FUNCTION_BLOCK Eventlogger
VAR
	Eventbuffer: ARRAY [1..MAXIMUM_NUMBER_OF_EVENTS] OF ST_Event;
	CurrentEventNumber : INT :=0;
	_PersistentEventStorage: I_PersistentStorage;
	
END_VAR
VAR CONSTANT
	MAXIMUM_NUMBER_OF_EVENTS: INT:=100;
END_VAR

METHOD PUBLIC AddEvent : BOOL
VAR_INPUT
	eEventType: E_EventType;
	eEventSeverity: TcEventSeverity;
	nEventIdentity: UDINT;
	sEventText: STRING(255);
END_VAR
IF NOT IsEventBufferFull() THEN
		CurrentEventNumber := CurrentEventNumber +1;
		Eventbuffer[CurrentEventNumber].eEventType:= eEventType;
		Eventbuffer[CurrentEventNumber].eEventSeverity:=eEventSeverity;
		Eventbuffer[CurrentEventNumber].nEventIdentity:=nEventIdentity;
		Eventbuffer[CurrentEventNumber].sEventText:=sEventText;
	UpdateEventTimeStampWithSystemTime(stEvent:= Eventbuffer[CurrentEventNumber]);	

AddEvent:=TRUE;
	ELSE
		AddEvent:=FALSE;	
	END_IF
	
	
	//Here we want to store the event persistently
	_PersistentEventStorage.StoreEvent(stEvent:=Eventbuffer[CurrentEventNumber]);
END_METHOD

METHOD FB_init : BOOL
VAR_INPUT
	bInitRetains : BOOL; // if TRUE, the retain variables are initialized (warm start / cold start)
	bInCopyCode : BOOL;  // if TRUE, the instance afterwards gets moved into the copy code (online change)
	iPersistentStorage: I_PersistentStorage;
	
END_VAR
_PersistentEventStorage:=iPersistentStorage;
END_METHOD

METHOD PRIVATE IsEventBufferFull : BOOL
VAR_INPUT
END_VAR
IsEventBufferFull:= (CurrentEventNumber+1 > MAXIMUM_NUMBER_OF_EVENTS);
END_METHOD

END_FUNCTION_BLOCK

(* stored: Version 1.1.0.1, ProductVersion 3.1.4024.11
   POU Eventlogger: Id {86ba1d44-1d92-4a05-b2ae-16ccae25a612}, SpecialFunc None
   Method AddEvent: Id {8871a3a6-8e53-472d-ad1f-4fddb60c1780}
   Method FB_init: Id {2ace2917-5694-4183-9366-d149fdcd0681}
   Method IsEventBufferFull: Id {65a64ffd-cabc-4ee7-b767-b780adb6ee79} *)
